// TIA Portal V17 export
// export: Created 2022-01-24T16:52:05.6528883Z, ExportSetting WithDefaults, DisplayName Totally Integrated Automation Portal, DisplayVersion V17, DisplayName TIA Portal Openness, DisplayVersion V17, DisplayName TIA Portal Version Control Interface, DisplayVersion V17, DisplayName SINAMICS Startdrive Advanced, DisplayVersion V17, DisplayName SINAMICS Startdrive G130, G150, S120, S150, SINAMICS MV, S210, DisplayVersion V17, DisplayName SINAMICS Startdrive G110M, G120, G120C, G120D, G120P, G115D, DisplayVersion V17, DisplayName STEP 7 Professional, DisplayVersion V17, DisplayName STEP 7 Safety, DisplayVersion V17, DisplayName WinCC Advanced, DisplayVersion V17
VAR_GLOBAL   // PLC tag table "Default tag table"
   Start AT %M0.0 : Bool;
   Rele AT %M10.0 : Bool;
   Tag_3 AT %M0.1 : Bool;
   Stop AT %M0.2 : Bool;
   stop2 AT %M0.3 : Bool;
   tlacStartM1 AT %I0.0 : Bool;
   tlacStopM1 AT %I10.0 : Bool;
   stykM1 AT %Q0.0 : Bool;
END_VAR
